ACTION IOFilter_action:
;
(* Update Functions for pin 1.2 *)
     (* Debounce filtering to raw DI value *)
     {{diX1_2_DebounceFb.name}}(i_In:={{diX1_2DiRaw.name}}, i_Delay:={{diX1_2_DebounceDelay.value}});
     {{diX1_2DiFiltered.name}} := {{diX1_2_DebounceFb.name}}.o_Out;
(* Update Functions for pin 1.3 *)
     (* Debounce filtering to raw DI value *)
     {{diX1_3_DebounceFb.name}}(i_In:={{diX1_3DiRaw.name}}, i_Delay:={{diX1_3_DebounceDelay.value}});
     {{diX1_3DiFiltered.name}} := {{diX1_3_DebounceFb.name}}.o_Out;
(* Update Functions for pin 1.7 *)
     (* Debounce filtering to raw DI value *)
     {{diX1_7_DebounceFb.name}}(i_In:={{diX1_7DiRaw.name}}, i_Delay:={{diX1_7_DebounceDelay.value}});
     {{diX1_7DiFiltered.name}} := {{diX1_7_DebounceFb.name}}.o_Out;
(* Update Functions for pin 1.8 *)
     (* Debounce filtering to raw DI value *)
     {{diX1_8_DebounceFb.name}}(i_In:={{diX1_8DiRaw.name}}, i_Delay:={{diX1_8_DebounceDelay.value}});
     {{diX1_8DiFiltered.name}} := {{diX1_8_DebounceFb.name}}.o_Out;
(* Update Functions for pin 1.9 *)
     (* Debounce filtering to raw DI value *)
     {{diX1_9_DebounceFb.name}}(i_In:={{diX1_9DiRaw.name}}, i_Delay:={{diX1_9_DebounceDelay.value}});
     {{diX1_9DiFiltered.name}} := {{diX1_9_DebounceFb.name}}.o_Out;
(* Update Functions for pin 1.10 *)
     (* Debounce filtering to raw DI value *)
     {{diX1_10_DebounceFb.name}}(i_In:={{diX1_10DiRaw.name}}, i_Delay:={{diX1_10_DebounceDelay.value}});
     {{diX1_10DiFiltered.name}} := {{diX1_10_DebounceFb.name}}.o_Out;
(* Update Functions for pin 1.11 *)
     (* Debounce filtering to raw DI value *)
     {{diX1_11_DebounceFb.name}}(i_In:={{diX1_11DiRaw.name}}, i_Delay:={{diX1_11_DebounceDelay.value}});
     {{diX1_11DiFiltered.name}} := {{diX1_11_DebounceFb.name}}.o_Out;
(* Update Functions for pin 1.12 *)
     (* Debounce filtering to raw DI value *)
     {{diX1_12_DebounceFb.name}}(i_In:={{diX1_12DiRaw.name}}, i_Delay:={{diX1_12_DebounceDelay.value}});
     {{diX1_12DiFiltered.name}} := {{diX1_12_DebounceFb.name}}.o_Out;
(* Update Functions for pin 1.14 *)
     (* Debounce filtering to raw DI value *)
     {{diX1_14_DebounceFb.name}}(i_In:={{diX1_14DiRaw.name}}, i_Delay:={{diX1_14_DebounceDelay.value}});
     {{diX1_14DiFiltered.name}} := {{diX1_14_DebounceFb.name}}.o_Out;
(* Update Functions for pin 1.15 *)
     (* Debounce filtering to raw DI value *)
     {{diX1_15_DebounceFb.name}}(i_In:={{diX1_15DiRaw.name}}, i_Delay:={{diX1_15_DebounceDelay.value}});
     {{diX1_15DiFiltered.name}} := {{diX1_15_DebounceFb.name}}.o_Out;
(* Make mean filtering for pin 1.20 *)

(* Make mean filtering for pin 1.20 *)

(* Make mean filtering for pin 1.21 *)

(* Make mean filtering for pin 1.20 *)

(* Filter actions for pin 1.22 *)
    {{aiX1_22AiFiltArrayIndex.name}}:= WORD_TO_BYTE({{aiX1_22AiFiltFb.name}}.o_Write);
    {{aiX1_22AiVarLatest.name}} := {{aiX1_22AiFiltArray.name}}[{{aiX1_22AiFiltArrayIndex.name}}];
    {{aiX1_22AiVarFilt.name}}:=AI_MeanValue(
        i_LatestBufferIndex := {{aiX1_22AiFiltArrayIndex.name}},
        i_pBuffer := {{aiX1_22AiFiltFb.name}}.i_Data,
        i_FirstIndex := 0,
        i_SizeOfBuffer := 50,
        i_Samples := {{aiX1_22AiFiltSamp.value}});
(* Filter actions for pin 1.23 *)
    {{aiX1_23AiFiltArrayIndex.name}}:= WORD_TO_BYTE({{aiX1_23AiFiltFb.name}}.o_Write);
    {{aiX1_23AiVarLatest.name}} := {{aiX1_23AiFiltArray.name}}[{{aiX1_23AiFiltArrayIndex.name}}];
    {{aiX1_23AiVarFilt.name}}:=AI_MeanValue(
        i_LatestBufferIndex := {{aiX1_23AiFiltArrayIndex.name}},
        i_pBuffer := {{aiX1_23AiFiltFb.name}}.i_Data,
        i_FirstIndex := 0,
        i_SizeOfBuffer := 50,
        i_Samples := {{aiX1_23AiFiltSamp.value}});
(* Update Functions for pin 1.25 *)
     (* Debounce filtering to raw DI value *)
     {{diX1_25_DebounceFb.name}}(i_In:={{diX1_25DiRaw.name}}, i_Delay:={{diX1_25_DebounceDelay.value}});
     {{diX1_25DiFiltered.name}} := {{diX1_25_DebounceFb.name}}.o_Out;
(* Update Functions for pin 1.26 *)
     (* Debounce filtering to raw DI value *)
     {{diX1_26_DebounceFb.name}}(i_In:={{diX1_26DiRaw.name}}, i_Delay:={{diX1_26_DebounceDelay.value}});
     {{diX1_26DiFiltered.name}} := {{diX1_26_DebounceFb.name}}.o_Out;
(* Update Functions for pin 1.27 *)
     (* Debounce filtering to raw DI value *)
     {{diX1_27_DebounceFb.name}}(i_In:={{diX1_27DiRaw.name}}, i_Delay:={{diX1_27_DebounceDelay.value}});
     {{diX1_27DiFiltered.name}} := {{diX1_27_DebounceFb.name}}.o_Out;
(* Make mean filtering for pin 1.31 *)

(* Make mean filtering for pin 1.20 *)

(* Make mean filtering for pin 1.32 *)

(* Make mean filtering for pin 1.20 *)

(* Filter actions for pin 1.34 *)
    {{aiX1_34AiFiltArrayIndex.name}}:= WORD_TO_BYTE({{aiX1_34AiFiltFb.name}}.o_Write);
    {{aiX1_34AiVarLatest.name}} := {{aiX1_34AiFiltArray.name}}[{{aiX1_34AiFiltArrayIndex.name}}];
    {{aiX1_34AiVarFilt.name}}:=AI_MeanValue(
            i_LatestBufferIndex := {{aiX1_34AiFiltArrayIndex.name}},
            i_pBuffer := {{aiX1_34AiFiltFb.name}}.i_Data,
            i_FirstIndex := 0,
            i_SizeOfBuffer := 50,
            i_Samples := {{aiX1_34AiFiltSamp.value}});
(* Filter actions for pin 1.35 *)
    {{aiX1_35AiFiltArrayIndex.name}}:= WORD_TO_BYTE({{aiX1_35AiFiltFb.name}}.o_Write);
    {{aiX1_35AiVarLatest.name}} := {{aiX1_35AiFiltArray.name}}[{{aiX1_35AiFiltArrayIndex.name}}];
    {{aiX1_35AiVarFilt.name}}:=AI_MeanValue(
             i_LatestBufferIndex := {{aiX1_35AiFiltArrayIndex.name}},
             i_pBuffer := {{aiX1_35AiFiltFb.name}}.i_Data,
             i_FirstIndex := 0,
             i_SizeOfBuffer := 50,
             i_Samples := {{aiX1_35AiFiltSamp.value}});
(* Update Functions for pin 1.2 *)
(* Update Functions for pin 1.3 *)
(* Update Functions for pin 1.7 *)
(* Update Functions for pin 1.8 *)
(* Update Functions for pin 1.14 *)
     (* Debounce filtering to raw DI value *)
     G_DebounceDI_SW_FOOT(i_In:=DI_RAW_SW_FOOT, i_Delay:=30);
     DI_SW_FOOT := G_DebounceDI_SW_FOOT.o_Out;
(* Update Functions for pin 1.15 *)
     (* Debounce filtering to raw DI value *)
     G_DebounceDI_SW_EMERGENCY(i_In:=DI_RAW_SW_EMERGENCY, i_Delay:=30);
     DI_SW_EMERGENCY := G_DebounceDI_SW_EMERGENCY.o_Out;
(* Make mean filtering for pin 1.20 *)

AI_ARR_INDEX_JOYSTICK_MV:= WORD_TO_BYTE(G_AIBufferOf_JOYSTICK_MV.o_Write);
AI_JOYSTICK_MV:=AI_MeanValue(
	i_LatestBufferIndex := AI_ARR_INDEX_JOYSTICK_MV,
	i_pBuffer := G_AIBufferOf_JOYSTICK_MV.i_Data,
	i_FirstIndex := 0,
	i_SizeOfBuffer := 50,
	i_Samples := 10);

(* Make mean filtering for pin 1.21 *)

AI_ARR_INDEX_SENSOR_MV:= WORD_TO_BYTE(G_AIBufferOf_SENSOR_MV.o_Write);
AI_SENSOR_MV:=AI_MeanValue(
	i_LatestBufferIndex := AI_ARR_INDEX_SENSOR_MV,
	i_pBuffer := G_AIBufferOf_SENSOR_MV.i_Data,
	i_FirstIndex := 0,
	i_SizeOfBuffer := 50,
	i_Samples := 10);

(* Filter actions for pin 1.22 *)
    AI_ARR_INDEX_VALVE_UPDN_CURRENT:= WORD_TO_BYTE(G_AIBufferOf_VALVE_UPDN_CURRENT.o_Write);
    FB_RAW_VALVE_UPDN_CURRENT := AI_ARR_VALVE_UPDN_CURRENT[AI_ARR_INDEX_VALVE_UPDN_CURRENT];
    FB_VALVE_UPDN_CURRENT:=AI_MeanValue(
        i_LatestBufferIndex := AI_ARR_INDEX_VALVE_UPDN_CURRENT,
        i_pBuffer := G_AIBufferOf_VALVE_UPDN_CURRENT.i_Data,
        i_FirstIndex := 0,
        i_SizeOfBuffer := 50,
        i_Samples := 10);
END_ACTION

ACTION Bus_action:
;
END_ACTION
END_ACTION

ACTION Application_action:
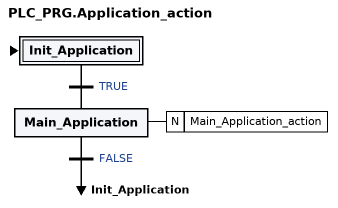
[picture p3: PLC_PRG.Application_action (SFC)]
INITIAL_STEP Init_Application:
END_STEP
TRANSITION FROM Init_Application TO Main_Application := TRUE;
END_TRANSITION
STEP Main_Application:
	Main_Application_action(N);
END_STEP
TRANSITION FROM Main_Application TO Init_Application := FALSE;
END_TRANSITION

ACTION Main_Application_action:
(* Call user application *)
    Main();
END_ACTION
END_ACTION

ACTION Epec_Out_action:
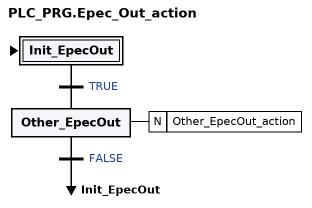
INITIAL_STEP Init_EpecOut:
END_STEP
TRANSITION FROM Init_EpecOut TO Other_EpecOut := TRUE;
END_TRANSITION
STEP Other_EpecOut:
	Other_EpecOut_action(N);
END_STEP
TRANSITION FROM Other_EpecOut TO Init_EpecOut := FALSE;
END_TRANSITION

ACTION Other_EpecOut_action:
NvRam_3606_Save();

IF NvRam_3606_Save.o_Busy = FALSE THEN
	SaveOdBlockActions(i_StateForActions := FALSE);
END_IF

(* Check reset request only if there is no data store going on. Exception is if error counter is bigger than 10 *)
IF G_RESET_MODULE AND NvRam_3606_Save.o_Busy = FALSE THEN
	(* Reset control unit *)
	SYSTEM_RESTART_PLCOPEN_APP(0);
END_IF

(* Block actions if voltage level is under defined limit *)
IF G_HWDiagnostics.o_SupplyVoltage > G_LowLimitForParameterSaving THEN

    (* Check if fast parameters are necessary to save *)
    IF G_3606_FastParamsSave = TRUE AND NvRam_3606_Save.o_Busy = FALSE THEN
        G_3606_FastParamsSave := FALSE;
        NvRam_3606_Save(
            i_SaveFastParamsStart:= TRUE,
            i_TimeOutValue:= G_3606_NVRAM_SAVE_MAX_TIME,
            i_SizeOfParams := G_3606_PARAM_SIZE,
            i_SizeOfFastParams := G_3606_FAST_PARAM_SIZE);
    END_IF

    (* If RAM image is changed nvram copying is always started again from begin. *)
    IF G_3606_OldImageChanged <> G_FileSysFileSystem.RamImageChanged AND G_3606_CopyNvRam.o_Busy = FALSE THEN
        SaveOdBlockActions(i_StateForActions := TRUE);
        G_3606_OldImageChanged := G_FileSysFileSystem.RamImageChanged;
        NvRam_3606_Save(
            i_SaveParamsStart:= TRUE,
            i_TimeOutValue:= G_3606_NVRAM_SAVE_MAX_TIME,
            i_SizeOfParams := G_3606_PARAM_SIZE,
            i_SizeOfFastParams := G_3606_FAST_PARAM_SIZE);
    END_IF

    (* Check if it is necessary to save communication parameters *)
    IF G_3606_CommsSaveOldCnt <> G_ODSAVE_SAVE_COMMS_COUNTER THEN
    ¤#COMM_CONFIGURATION#1#¤
        SystemParameters.WriteData();
        G_3606_CommsSaveOldCnt := G_ODSAVE_SAVE_COMMS_COUNTER;
    END_IF

    (* Check if it is necessary to restor communication parameters *)
    IF G_3606_CommsRestoreOldCnt <> G_ODSAVE_RESTORE_COMMS_COUNTER THEN
        (* Restore communication parameters *)
        SystemParameters.RestoreDefaultData();
    ¤#COMM_CONFIGURATION#0#¤
        G_3606_CommsRestoreOldCnt := G_ODSAVE_RESTORE_COMMS_COUNTER;
    END_IF

END_IF
    
(* Overcurrent protection for mA AI inputs *)
AIP_InputProtection_3606(
	o_NoErrors=>G_NoErrors ,
	o_XM1_20_OverCurrent=>G_X1_20_OverCurrent ,
	o_XM1_21_OverCurrent=>G_X1_21_OverCurrent ,
	o_XM1_31_OverCurrent=>G_X1_31_OverCurrent,
	o_XM1_32_OverCurrent=>G_X1_32_OverCurrent );
END_ACTION
END_ACTION
END_PROGRAM
